FUNCTION "FC_Dereg_LNK_In_PLT" : VOID
TITLE =%version: 1.06 % CN: 33
//Function:
//This FC removes a LNK and LIC from the PLT DB and sends a Deregister.
//
//
//                       Downstream PLT DB
// IF Down present       ______
// Check First entry     |    v
//        ____________________________________
//                         |
//   ===flow-direction===> |
//        TRS xx           |
//        _________________|__________________
//
// IF No Down present     ^
//                        |
//             Read pos = 0 + max dis
//
//Description:
//When an Leading edge is found in first entry with data, this data (LNK and LIC)
//is deassigned
//and a Deregister is send.
//
//History:
//This version  %created_by:  nlhdl %
//              %date_created:  maandag 6 juli 2015 10:33:09 %
//              %release:  VI_CONV/RA_Dev_Oakham %
//
//Modification History:                                   By:    Date:     Rev:
//----------------------------------------------------  -------  --------  -----
//7324: ECS-P General from the RD to RA for platform    nlHdL    06-07-15   1.06
//22337: Remove the vibes1.x with the vibes 3.x         nlHdL    09-01-15   1.06
//19518: Block call update of FC_xxx_Record             nltny    07-08-14   0.02
//Initial Version based on version 1.04 ECS-P GEN       nlHHop   01-04-14   0.01
//
FAMILY : VIBES
VERSION : 0.0


VAR_INPUT
  i_DB_PLT_Num : INT ;	//Number of DB Position Leading Trailing Edge
  i_DB_Event_Num : INT ;	//Number of DB event
  i_Arrived_Position : INT ;	//Location number of where bag is end of tracking
END_VAR
VAR_TEMP
  t_DB_PLT : INT ;	//Number of PLT DB
  t_position : INT ;	//Position entry in PLT DB
  t_Info : INT ;	//Info entry in PLT DB
  t_Data : INT ;	//Data entry in PLT DB
  t_DB_Event_Nr : INT ;	//Number of DB Event
  t_Return_Value_Int : INT ;	//Dummy return value
  t_ECS : INT ;	//ECS number of generated LNK
END_VAR
BEGIN
NETWORK
TITLE =AA: Read DB info and PLT

      L     #i_DB_Event_Num;
      T     #t_DB_Event_Nr;

      L     #i_DB_PLT_Num;
      T     #t_DB_PLT; // Determine PLT block DB number

      OPN   DB [#t_DB_PLT];

      AN    DBX   10.1; // Conveyor is NOT running stop block.
      BEC   ;

      L     DBW    8;
      L     1;
      >I    ;
      JCN   AA01;

//Open Downstream PLT DB
      OPN   DB [DBW 8];

      L     DBW   14;
      T     #t_position;

      L     DBW   18;
      T     #t_Info;

      L     DBW   20;
      T     #t_Data;

// Remove the LNK number
      L     0;
      T     DBW   20;
      JU    AA99;

//IF No downstream read from position 0
AA01: CALL "FC_PLT_Srch_Win_Up" (
           i_DB_PLT_Num             := #t_DB_PLT,
           i_Position               := 1,// 1 cm before end of conveyor
           i_Window                 := 0,
           o_Position               := #t_position,
           o_Info                   := #t_Info,
           o_LNK                    := #t_Data,
           o_DB_PLT_Num             := #t_Return_Value_Int,
           o_Number_Items_Found     := #t_Return_Value_Int);

      CALL "FC_PLT_Clr_Position" (
           i_DB_PLT_Num             := #t_DB_PLT,
           i_Position               := #t_position,
           i_Info_Physical          := #t_Info,
           i_DB_Event_Num           := #t_DB_Event_Nr);

AA99: NOP   0;
NETWORK
TITLE =BA: Remove LNK in PLT and Deregister the LNK

      L     #t_Info;
      L     1;
      ==I   ;
      JCN   BA99;

      L     #t_Data;
      L     0;
      <>I   ;
      JCN   BA99;

// Read ECS number in LNK DB
      CALL "FC_Read_Int_Record" (
           i_Record_Number          := #t_Data,
           i_P_INT_Record           := "DB_UDT_LNK_Record".ECS,
           i_DB                     := "DB_LNK_List",
           i_DB_Event_Num           := #t_DB_Event_Nr,
           o_INT                    := #t_ECS);

      L     #t_ECS;
      L     0;
      >I    ;
      JCN   BA99;

      CALL "FC_Write_Int_Record" (
           i_Record_Number          := #t_ECS,
           i_P_INT_Record           := "DB_UDT_ECS_Record".Routing_Result.Arrived_Location,
           i_DB                     := "DB_ECS_List",
           i_INT                    := #i_Arrived_Position,
           i_DB_Event_Num           := #t_DB_Event_Nr);

      CALL "FC_Write_Event" (// Package report "Arrived"
           i_Message_ID             := 1211,
           i_Event_value            := #t_Data,
           i_DB_Event_Num           := #t_DB_Event_Nr,
           o_Return_Value           := #t_Return_Value_Int);

// Write correct deregister reason in CIR
      CALL "FC_Write_BOOL_Record" (
           i_Record_Number          := #t_ECS,
           i_P_BOOL_Record          := "DB_UDT_ECS_Record".CIR.Expected_Item,
           i_DB                     := "DB_ECS_List",
           i_BOOL                   := TRUE,
           i_DB_Event_Num           := #t_DB_Event_Nr);

      CALL "FC_Write_BOOL_Record" (
           i_Record_Number          := #t_ECS,
           i_P_BOOL_Record          := "DB_UDT_ECS_Record".CIR.Unexpected_Item,
           i_DB                     := "DB_ECS_List",
           i_BOOL                   := FALSE,
           i_DB_Event_Num           := #t_DB_Event_Nr);

      CALL "FC_Write_BOOL_Record" (
           i_Record_Number          := #t_ECS,
           i_P_BOOL_Record          := "DB_UDT_ECS_Record".CIR.Hand_Over,
           i_DB                     := "DB_ECS_List",
           i_BOOL                   := FALSE,
           i_DB_Event_Num           := #t_DB_Event_Nr);

      CALL "FC_Write_Event" (// Report Deregisterpackage (1206)
           i_Message_ID             := 1206,
           i_Event_value            := #t_Data,
           i_DB_Event_Num           := #t_DB_Event_Nr,
           o_Return_Value           := #t_Return_Value_Int);

BA99: NOP   0;
END_FUNCTION

